PROGRAM commandExecute
VAR
	MCPower_Xa, MCPower_Xb, MCPower_Y, 	MCPower_Z 	: MC_Power;
	MCResetXa, MCResetXb, MCResetY, MCResetZ		: MC_Reset;

	fb_MCGearIn										: MC_GearIn;
	fb_MCGearOut									: MC_GearOut;

	fb_MCHOME_X, fb_MCHOME_Y						: MC_Home;
	fb_MoveAbs_X, fb_MoveAbs_Y, fb_MoveAbs_Z 		: MC_MoveAbsolute;
	fb_MoveRel_Z 									: MC_MoveRelative;
	fb_ReadX, fb_ReadY, fb_readZ 					: MC_ReadActualPosition;

	fb_SetZToZero 									: MC_SetPosition;
END_VAR

//Enable Axis
	MCPower_Xa(
		Axis	:= GVL.As_Xa, 
		Enable	:= COM.bEnable, 
		Enable_Positive:= COM.bEnable, 
		Enable_Negative:= COM.bEnable, 
		Override:= 100 );
		
	MCPower_Xb(
		Axis	:= GVL.As_Xb, 
		Enable	:= COM.bEnable, 
		Enable_Positive:= COM.bEnable, 
		Enable_Negative:= COM.bEnable, 
		Override:= 100 );
		
	MCPower_Y(
		Axis	:= GVL.As_Y, 
		Enable	:= COM.bEnable, 
		Enable_Positive:= COM.bEnable, 
		Enable_Negative:= COM.bEnable, 
		Override:= 100 );
		
	MCPower_Z(
		Axis	:= GVL.As_Z, 
		Enable	:= COM.bEnable, 
		Enable_Positive:= COM.bEnable, 
		Enable_Negative:= COM.bEnable, 
		Override:= 100 );

//Reset Axis
	MCResetXa(
		Axis	:= GVL.As_Xa, 
		Execute	:= COM.bReset );
	
	MCResetXb(
		Axis	:= GVL.As_Xb, 
		Execute	:= COM.bReset );

	MCResetY(
		Axis	:= GVL.As_Y, 
		Execute	:= COM.bReset );

	MCResetZ(
		Axis	:= GVL.As_Z, 
		Execute	:= COM.bReset );
	
//Couple Axis
	fb_MCGearIn(
		Master	:= GVL.As_Xa, 
		Slave	:= GVL.As_Xb, 
		Execute := COM.bCouple, 
		RatioNumerator:= 1, 
		RatioDenominator:= 1 );
		
	fb_MCGearOut(
		Slave	:= GVL.As_Xb,
		Execute := NOT(COM.bCouple) );
		
//Homing
	fb_MCHOME_X(
		Axis     := GVL.As_Xa, 
		Execute  := COM.bHome AND COM.bCouple, 
		Position := 0, 
		bCalibrationCam:= GVL.bX1 );
	
	fb_MCHOME_Y(
		Axis	 := GVL.As_Y, 
		Execute  := COM.bHome AND COM.bCouple, 
		Position := 0, 
		bCalibrationCam:= GVL.bY1 );
		
//Absolute movement
	fb_MoveAbs_X(
		Axis 	 := GVL.As_Xa,
		Execute  := COM.bMoveX AND COM.bCouple,
		Position := COM.absX,
		Velocity := COM.velX);
		
	fb_MoveAbs_Y(
		Axis 	 := GVL.As_Y,
		Execute  := COM.bMoveY,
		Position := COM.absY,
		Velocity := COM.velY);		
		
	fb_MoveAbs_Z(
		Axis 	 := GVL.As_Z,
		Execute  := COM.bMoveZ,
		Position := COM.absZ,
		Velocity := COM.velZ);
//Rel movement
	fb_MoveRel_Z(
		Axis 	 := GVL.As_Z,
		Execute  := COM.bRelZ,
		distance := COM.relZ,
		Velocity := COM.velZ);			
		
//set Z postition to zero
	fb_SetZToZero(
		Axis := GVL.As_Z, 
		Execute := COM.bSetZ,
		Position := 0, 
		Mode := FALSE);

//read actual position
	fb_ReadX(Enable := TRUE, Axis := GVL.As_Xa, Position => COM.PosX);
	fb_ReadY(Enable := TRUE, Axis := GVL.As_Y, Position => COM.PosY);
	fb_ReadZ(Enable := TRUE, Axis := GVL.As_Z, Position => COM.PosZ);
	COM.bValid := fb_ReadX.Valid AND fb_ReadY.Valid AND fb_ReadZ.Valid;
	
//done = busy
	COM.bHomeBusy	:= fb_MCHOME_X.Busy OR fb_MCHOME_Y.Busy;
	COM.bMoveBusy	:= fb_MoveAbs_X.Busy OR fb_MoveAbs_Y.Busy OR fb_MoveAbs_Z.Busy;		
	
	COM.bHomeDone	:= fb_MCHOME_X.Done AND fb_MCHOME_Y.Done;
	COM.bMoveDone	:= fb_MoveAbs_X.Done AND fb_MoveAbs_Y.Done AND fb_MoveAbs_Z.Done;
	
	COM.bMoveXDone	:= fb_MoveAbs_X.Done;
	COM.bMoveYDone	:= fb_MoveAbs_Y.Done;
	COM.bMoveZDone	:= fb_MoveAbs_Z.Done;
	COM.bMoveZRelDone	:= fb_MoveRel_Z.Done;

END_PROGRAM

(* stored: Version 1.1.0.1, ProductVersion 3.1.4024.2
   POU commandExecute: Id {4ff840c8-9717-45e8-bdfc-1a7c01fc0485}, SpecialFunc None *)
